Omron CX-Programmer project NewProject (CX-Programmer 9.61)

# PLC NewPLC1: CP1E N20

## Global symbols (name address type ; comment)
0 CHANNEL  ; Stop Stepper
0.04 BOOL  ; En_Stepper1
0.05 BOOL  ; en Stepper2
200.00 BOOL  ; Stepper1_CCW
200.01 BOOL  ; Stepper1_CW
200.02 BOOL  ; Stop Stepper1
200.03 BOOL  ; Enable STepper 1
201.00 BOOL  ; Setepper2_CCW
201.01 BOOL  ; Stepper2_CW
201.03 BOOL  ; Enable Stepper1
D100 CHANNEL  ; Move Stepper
D110 CHANNEL  ; CCW
D200 CHANNEL  ; MOVE CCW

## Program NewProgram1 (cyclic task 0)

### Section Main

### Section Stepper1_Move

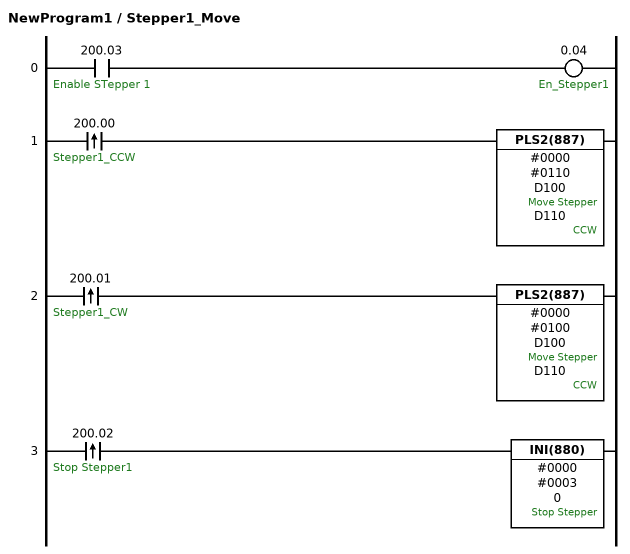
; rung 0
LD 200.03  ; Enable STepper 1
OUT 0.04  ; En_Stepper1
; rung 1
@LD 200.00  ; Stepper1_CCW
PLS2(887) #0000 #0110 D100 D110  ; Move Stepper, CCW
; rung 2
@LD 200.01  ; Stepper1_CW
PLS2(887) #0000 #0100 D100 D110  ; Move Stepper, CCW
; rung 3
@LD 200.02  ; Stop Stepper1
INI(880) #0000 #0003 0  ; Stop Stepper

### Section Stepper2_Move

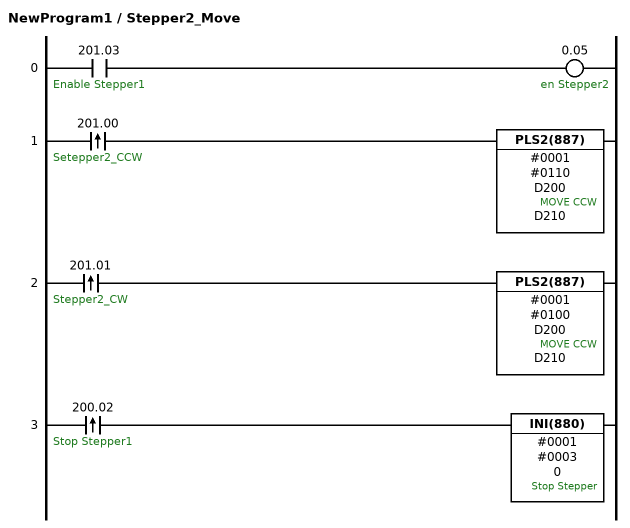
; rung 0
LD 201.03  ; Enable Stepper1
OUT 0.05  ; en Stepper2
; rung 1
@LD 201.00  ; Setepper2_CCW
PLS2(887) #0001 #0110 D200 D210  ; MOVE CCW
; rung 2
@LD 201.01  ; Stepper2_CW
PLS2(887) #0001 #0100 D200 D210  ; MOVE CCW
; rung 3
@LD 200.02  ; Stop Stepper1
INI(880) #0001 #0003 0  ; Stop Stepper

### Section END
; rung 0
END(001)